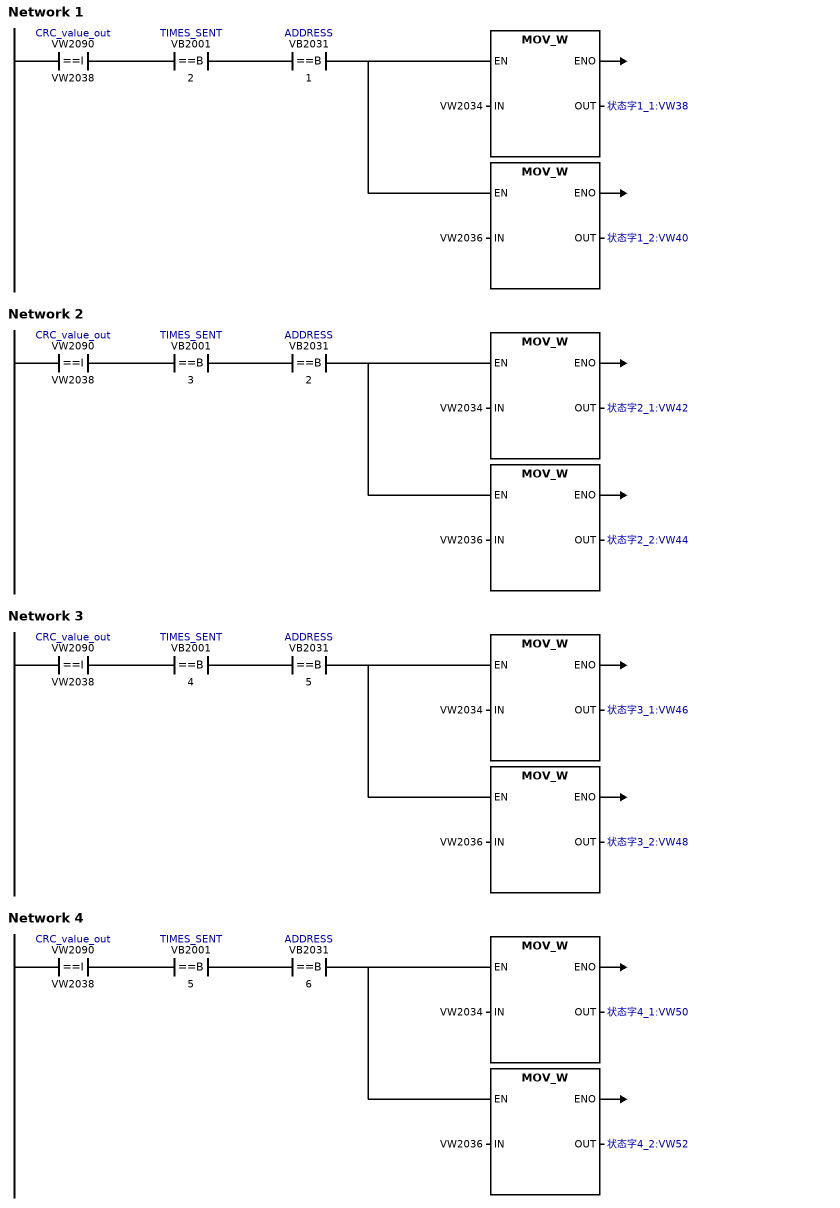
[picture p48: SBR52 networks 1-4]
Network 1
LDW=   CRC_value_out:VW2090, VW2038
AB=    TIMES_SENT:VB2001, 2
AB=    ADDRESS:VB2031, 1
MOVW   VW2034, 状态字1_1:VW38
MOVW   VW2036, 状态字1_2:VW40
Network 2
LDW=   CRC_value_out:VW2090, VW2038
AB=    TIMES_SENT:VB2001, 3
AB=    ADDRESS:VB2031, 2
MOVW   VW2034, 状态字2_1:VW42
MOVW   VW2036, 状态字2_2:VW44
Network 3
LDW=   CRC_value_out:VW2090, VW2038
AB=    TIMES_SENT:VB2001, 4
AB=    ADDRESS:VB2031, 5
MOVW   VW2034, 状态字3_1:VW46
MOVW   VW2036, 状态字3_2:VW48
Network 4
LDW=   CRC_value_out:VW2090, VW2038
AB=    TIMES_SENT:VB2001, 5
AB=    ADDRESS:VB2031, 6
MOVW   VW2034, 状态字4_1:VW50
MOVW   VW2036, 状态字4_2:VW52
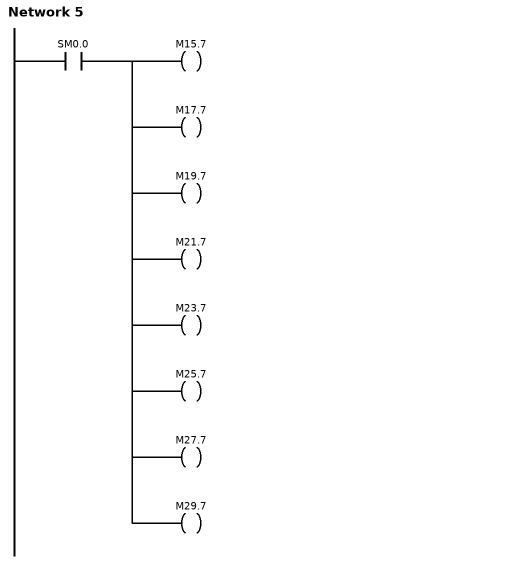
Network 5
LD     SM0.0
=      M15.7
=      M17.7
=      M19.7
=      M21.7
=      M23.7
=      M25.7
=      M27.7
=      M29.7
END_SUBROUTINE_BLOCK

SUBROUTINE_BLOCK COMM_CHECK:SBR53
TITLE=SUBROUTINE COMMENTS
VAR
TEMP1:BOOL;	// L0.0 
TEMP2:BOOL;	// L0.1 
TEMP3:BOOL;	// L0.2 
END_VAR
BEGIN
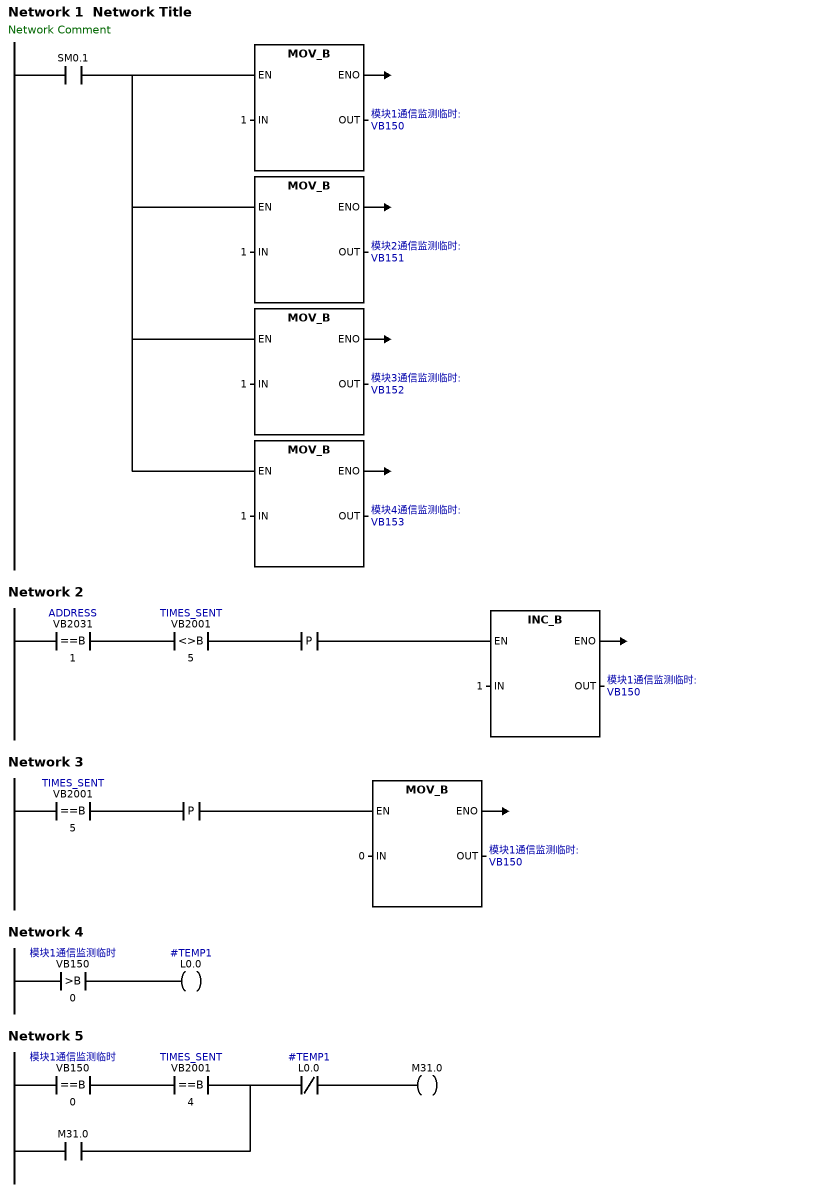
Network 1 // Network Title
// Network Comment
LD     SM0.1
MOVB   1, 模块1通信监测临时:VB150
MOVB   1, 模块2通信监测临时:VB151
MOVB   1, 模块3通信监测临时:VB152
MOVB   1, 模块4通信监测临时:VB153
Network 2
LDB=   ADDRESS:VB2031, 1
AB<>   TIMES_SENT:VB2001, 5
EU
MOVB   1, 模块1通信监测临时:VB150
INCB   模块1通信监测临时:VB150
Network 3
LDB=   TIMES_SENT:VB2001, 5
EU
MOVB   0, 模块1通信监测临时:VB150
Network 4
LDB>   模块1通信监测临时:VB150, 0
=      #TEMP1:L0.0
Network 5
LDB=   模块1通信监测临时:VB150, 0
AB=    TIMES_SENT:VB2001, 4
O      M31.0
AN     #TEMP1:L0.0
=      M31.0
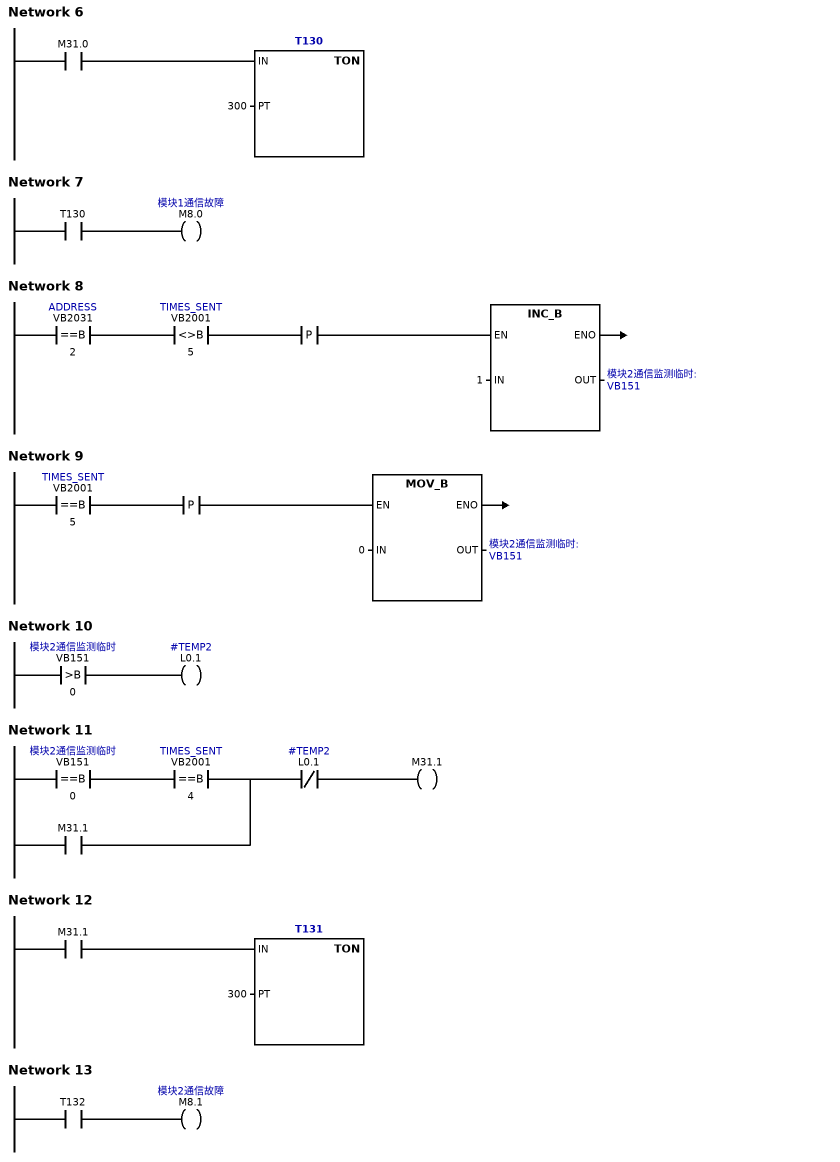
Network 6
LD     M31.0
TON    T130, 300
Network 7
LD     T130
=      模块1通信故障:M8.0
Network 8
LDB=   ADDRESS:VB2031, 2
AB<>   TIMES_SENT:VB2001, 5
EU
MOVB   1, 模块2通信监测临时:VB151
INCB   模块2通信监测临时:VB151
Network 9
LDB=   TIMES_SENT:VB2001, 5
EU
MOVB   0, 模块2通信监测临时:VB151
Network 10
LDB>   模块2通信监测临时:VB151, 0
=      #TEMP2:L0.1
Network 11
LDB=   模块2通信监测临时:VB151, 0
AB=    TIMES_SENT:VB2001, 4
O      M31.1
AN     #TEMP2:L0.1
=      M31.1
Network 12
LD     M31.1
TON    T131, 300
Network 13
LD     T132
=      模块2通信故障:M8.1
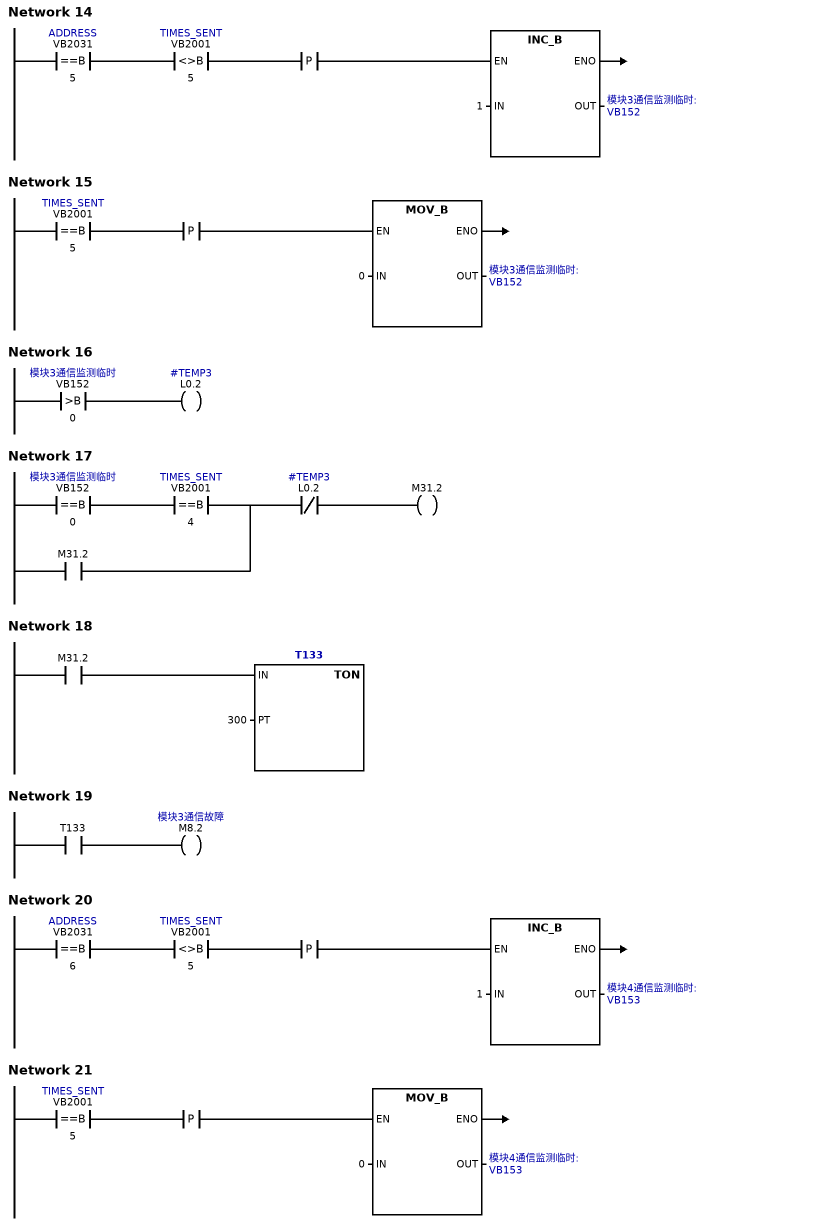
Network 14
LDB=   ADDRESS:VB2031, 5
AB<>   TIMES_SENT:VB2001, 5
EU
MOVB   1, 模块3通信监测临时:VB152
INCB   模块3通信监测临时:VB152
Network 15
LDB=   TIMES_SENT:VB2001, 5
EU
MOVB   0, 模块3通信监测临时:VB152
Network 16
LDB>   模块3通信监测临时:VB152, 0
=      #TEMP3:L0.2
Network 17
LDB=   模块3通信监测临时:VB152, 0
AB=    TIMES_SENT:VB2001, 4
O      M31.2
AN     #TEMP3:L0.2
=      M31.2
Network 18
LD     M31.2
TON    T133, 300
Network 19
LD     T133
=      模块3通信故障:M8.2
Network 20
LDB=   ADDRESS:VB2031, 6
AB<>   TIMES_SENT:VB2001, 5
EU
MOVB   1, 模块4通信监测临时:VB153
INCB   模块4通信监测临时:VB153
Network 21
LDB=   TIMES_SENT:VB2001, 5
EU
MOVB   0, 模块4通信监测临时:VB153
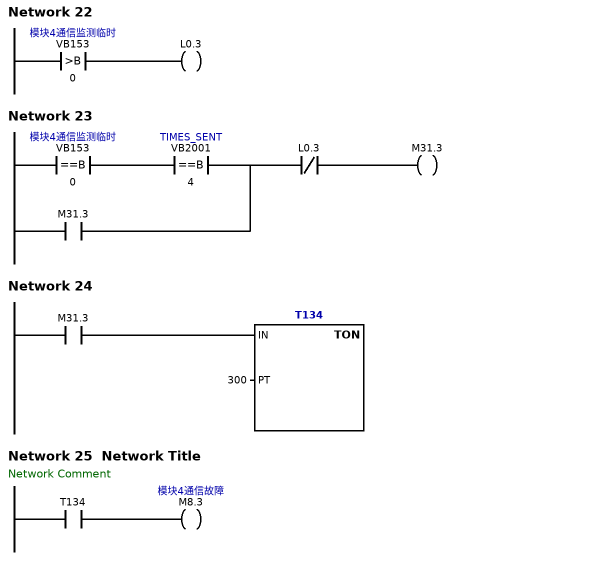
Network 22
LDB>   模块4通信监测临时:VB153, 0
=      L0.3
Network 23
LDB=   模块4通信监测临时:VB153, 0
AB=    TIMES_SENT:VB2001, 4
O      M31.3
AN     L0.3
=      M31.3
Network 24
LD     M31.3
TON    T134, 300
Network 25 // Network Title
// Network Comment
LD     T134
=      模块4通信故障:M8.3
END_SUBROUTINE_BLOCK

SUBROUTINE_BLOCK COMM_ARRAY:SBR54
TITLE=SUBROUTINE COMMENTS
VAR_INPUT
SLAVER_ADR:BYTE;	// LB0 
STAR_REG:BYTE;	// LB1 
REG_LEN:BYTE;	// LB2 
END_VAR
VAR_OUTPUT
ARRAY_T1:WORD;	// LW3 
ARRAY_T2:WORD;	// LW5 
ARRAY_T3:WORD;	// LW7 
ARRAY_T4:WORD;	// LW9 
END_VAR
BEGIN
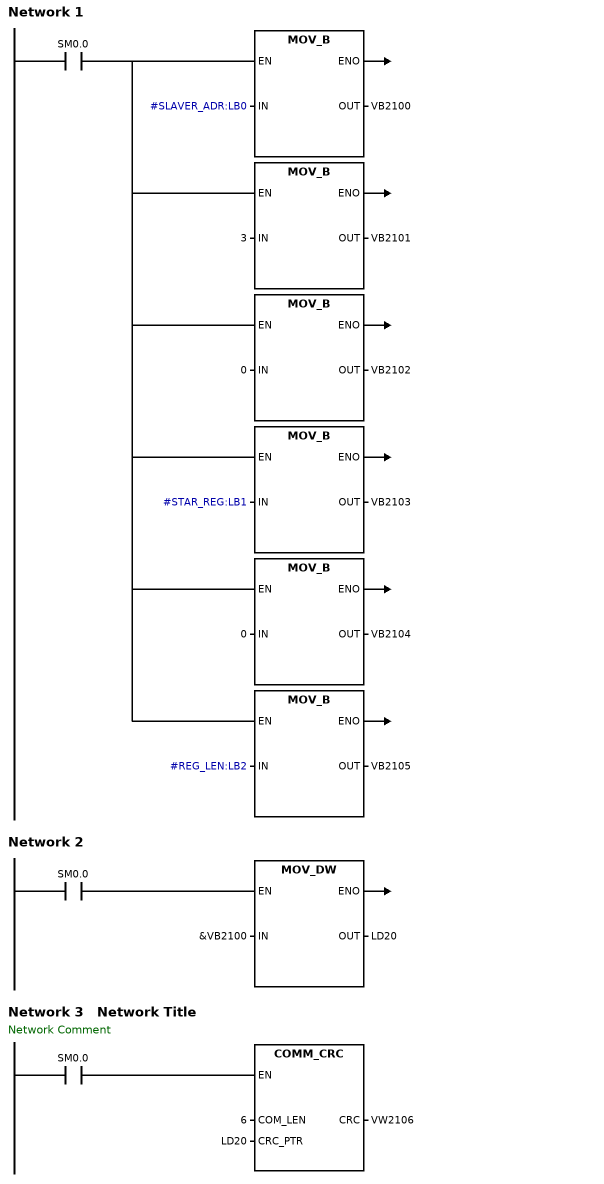
Network 1
LD     SM0.0
MOVB   #SLAVER_ADR:LB0, VB2100
MOVB   3, VB2101
MOVB   0, VB2102
MOVB   #STAR_REG:LB1, VB2103
MOVB   0, VB2104
MOVB   #REG_LEN:LB2, VB2105
Network 2
LD     SM0.0
MOVD   &VB2100, LD20
Network 3 //  Network Title
//  Network Comment
LD     SM0.0
CALL   COMM_CRC:SBR51, 6, LD20, VW2106
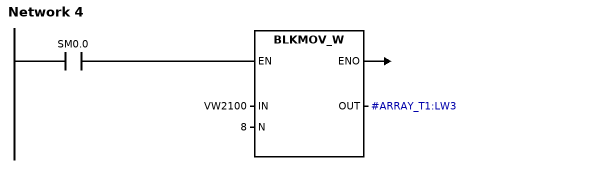
Network 4
LD     SM0.0
BMW    VW2100, #ARRAY_T1:LW3, 8
END_SUBROUTINE_BLOCK

SUBROUTINE_BLOCK PORT_SET:SBR55
TITLE=SUBROUTINE COMMENTS
VAR_INPUT
PORT:BYTE;	// LB0 端口
SPEECH:WORD;	// LW1 通信速率（1200，2400，4800，9600，19200）
DATABIT:BYTE;	// LB3 数据位（7或8）
CHECK:BYTE;	// LB4 是否校验（0：无校验；1：偶校验；2：奇校验）
END_VAR
VAR
ONN:BOOL;	// L5.0 
SETING:BYTE;	// LB6 
TEMP:WORD;	// LW7 
END_VAR
BEGIN
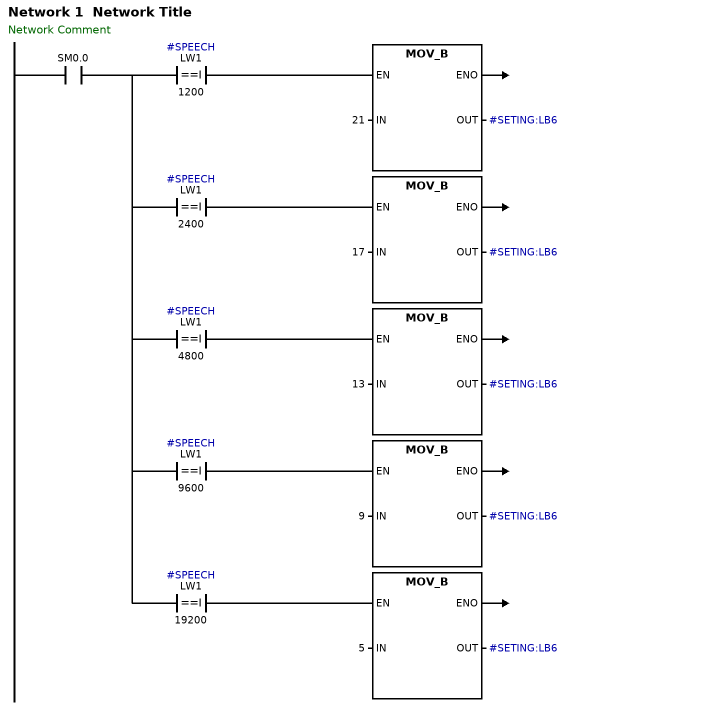
Network 1 // Network Title
// Network Comment
// (network saved uncompiled; LAD cells follow)
// row 0: c0 -| |- SM0.0 v  c1 -|==I|- #SPEECH:LW1, 1200  c2 --  c3 [MOV_B EN:=power@row0, IN:=21, ENO=>power, OUT=>#SETING:LB6]  c4 ->
// row 1: c0 ^v  c3 [box]
// row 2: c0 ^v  c1 -|==I|- #SPEECH:LW1, 2400  c2 --  c3 [MOV_B EN:=power@row2, IN:=17, ENO=>power, OUT=>#SETING:LB6]  c4 ->
// row 3: c0 ^v  c3 [box]
// row 4: c0 ^v  c1 -|==I|- #SPEECH:LW1, 4800  c2 --  c3 [MOV_B EN:=power@row4, IN:=13, ENO=>power, OUT=>#SETING:LB6]  c4 ->
// row 5: c0 ^v  c3 [box]
// row 6: c0 ^v  c1 -|==I|- #SPEECH:LW1, 9600  c2 --  c3 [MOV_B EN:=power@row6, IN:=9, ENO=>power, OUT=>#SETING:LB6]  c4 ->
// row 7: c0 ^v  c3 [box]
// row 8: c0 ^  c1 -|==I|- #SPEECH:LW1, 19200  c2 --  c3 [MOV_B EN:=power@row8, IN:=5, ENO=>power, OUT=>#SETING:LB6]  c4 ->
// row 9: c3 [box]
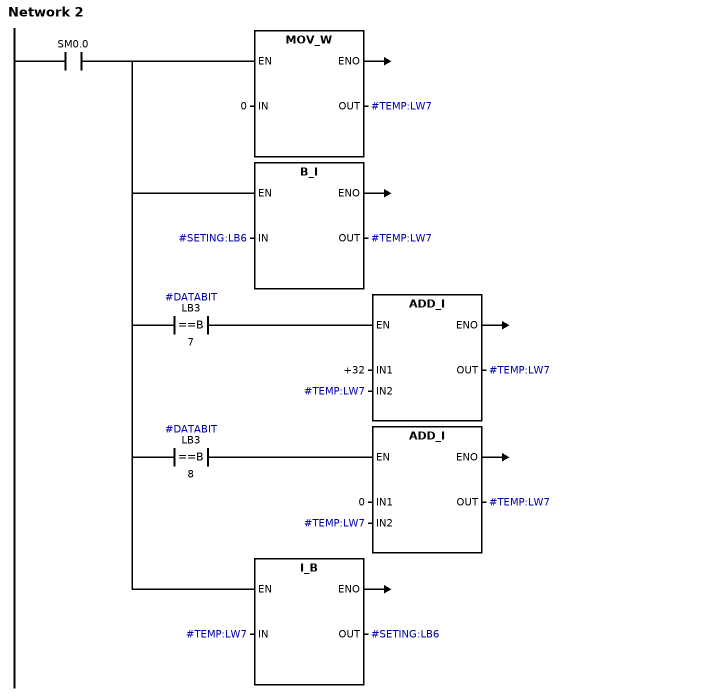
Network 2
// (network saved uncompiled; LAD cells follow)
// row 0: c0 -| |- SM0.0 v  c1 --  c2 [MOV_W EN:=power@row0, IN:=0, ENO=>power, OUT=>#TEMP:LW7]  c3 ->
// row 1: c0 ^v  c2 [box]
// row 2: c0 ^v  c1 --  c2 [B_I EN:=power@row2, IN:=#SETING:LB6, ENO=>power, OUT=>#TEMP:LW7]  c3 ->
// row 3: c0 ^v  c2 [box]
// row 4: c0 ^v  c1 -|==B|- #DATABIT:LB3, 7  c2 --  c3 [ADD_I EN:=power@row4, IN1:=+32, IN2:=#TEMP:LW7, ENO=>power, OUT=>#TEMP:LW7]  c4 ->
// row 5: c0 ^v  c3 [box]
// row 6: c0 ^v  c1 -|==B|- #DATABIT:LB3, 8  c2 --  c3 [ADD_I EN:=power@row6, IN1:=0, IN2:=#TEMP:LW7, ENO=>power, OUT=>#TEMP:LW7]  c4 ->
// row 7: c0 ^v  c3 [box]
// row 8: c0 ^  c1 --  c2 [I_B EN:=power@row8, IN:=#TEMP:LW7, ENO=>power, OUT=>#SETING:LB6]  c3 ->
// row 9: c2 [box]
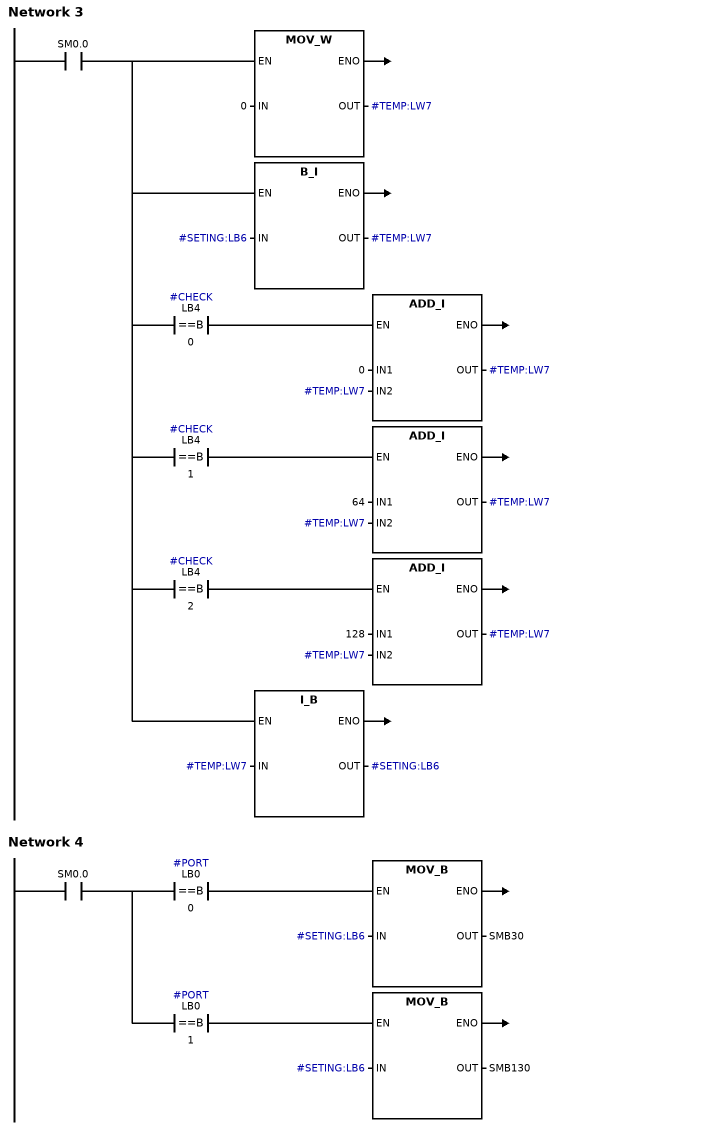
Network 3
// (network saved uncompiled; LAD cells follow)
// row 0: c0 -| |- SM0.0 v  c1 --  c2 [MOV_W EN:=power@row0, IN:=0, ENO=>power, OUT=>#TEMP:LW7]  c3 ->
// row 1: c0 ^v  c2 [box]
// row 2: c0 ^v  c1 --  c2 [B_I EN:=power@row2, IN:=#SETING:LB6, ENO=>power, OUT=>#TEMP:LW7]  c3 ->
// row 3: c0 ^v  c2 [box]
// row 4: c0 ^v  c1 -|==B|- #CHECK:LB4, 0  c2 --  c3 [ADD_I EN:=power@row4, IN1:=0, IN2:=#TEMP:LW7, ENO=>power, OUT=>#TEMP:LW7]  c4 ->
// row 5: c0 ^v  c3 [box]
// row 6: c0 ^v  c1 -|==B|- #CHECK:LB4, 1  c2 --  c3 [ADD_I EN:=power@row6, IN1:=64, IN2:=#TEMP:LW7, ENO=>power, OUT=>#TEMP:LW7]  c4 ->
// row 7: c0 ^v  c3 [box]
// row 8: c0 ^v  c1 -|==B|- #CHECK:LB4, 2  c2 --  c3 [ADD_I EN:=power@row8, IN1:=128, IN2:=#TEMP:LW7, ENO=>power, OUT=>#TEMP:LW7]  c4 ->
// row 9: c0 ^v  c3 [box]
// row 10: c0 ^  c1 --  c2 [I_B EN:=power@row10, IN:=#TEMP:LW7, ENO=>power, OUT=>#SETING:LB6]  c3 ->
// row 11: c2 [box]
Network 4
// (network saved uncompiled; LAD cells follow)
// row 0: c0 -| |- SM0.0 v  c1 -|==B|- #PORT:LB0, 0  c2 --  c3 [MOV_B EN:=power@row0, IN:=#SETING:LB6, ENO=>power, OUT=>SMB30]  c4 ->
// row 1: c0 ^v  c3 [box]
// row 2: c0 ^  c1 -|==B|- #PORT:LB0, 1  c2 --  c3 [MOV_B EN:=power@row2, IN:=#SETING:LB6, ENO=>power, OUT=>SMB130]  c4 ->
// row 3: c3 [box]
END_SUBROUTINE_BLOCK

SUBROUTINE_BLOCK MES_SEND:SBR56
TITLE=SUBROUTINE COMMENTS
BEGIN
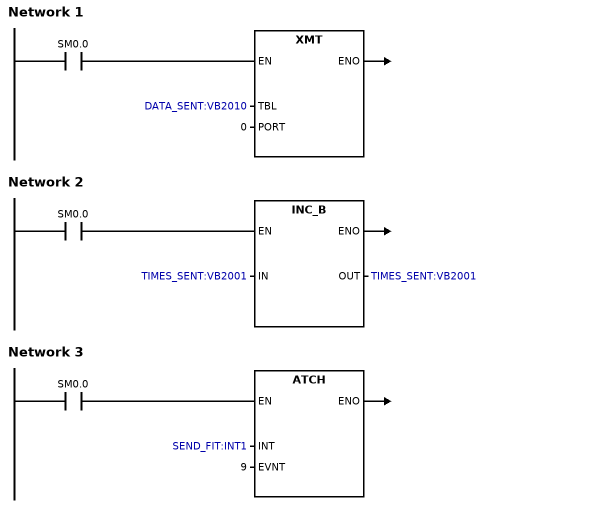
Network 1 // 
	
LD     SM0.0
XMT    DATA_SENT:VB2010, 0
Network 2
LD     SM0.0
INCB   TIMES_SENT:VB2001
Network 3
LD     SM0.0
ATCH   SEND_FIT:INT1, 9
Network 4 // Network Title
// Network Comment
END_SUBROUTINE_BLOCK

SUBROUTINE_BLOCK ARRAY_INSTR:SBR60
TITLE=旧的4块镇流器监测模块的地址分别是1,2,3,5
BEGIN
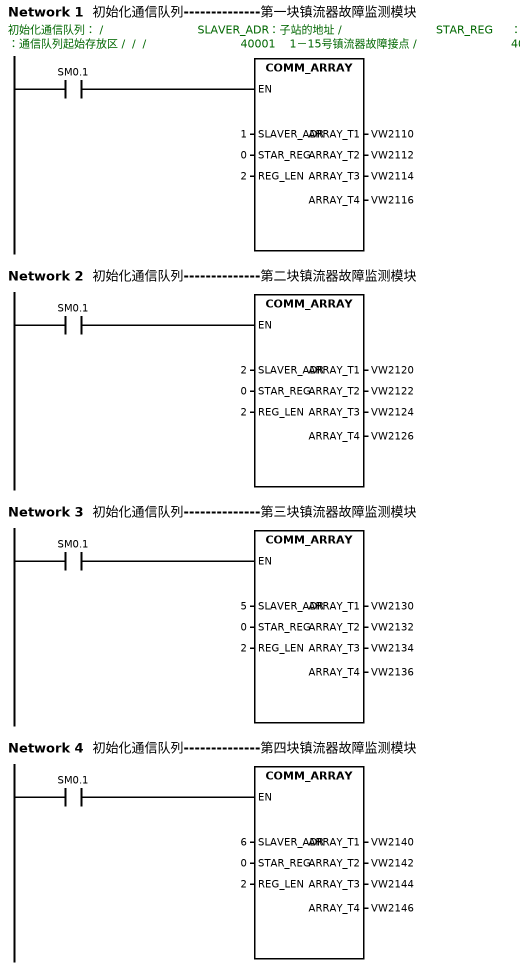
Network 1 // 初始化通信队列--------------第一块镇流器故障监测模块
// 初始化通信队列：
//                           SLAVER_ADR：子站的地址
//                           STAR_REG     ：子站数据起始寄存器
//                           REG_LEN        ：读取的数据寄存器长度
//                           ARRAY_T        ：通信队列起始存放区
// 
// 
//                           40001		1－15号镇流器故障接点
//                           40002		16－30号镇流器故障接点
//                         
LD     SM0.1
CALL   COMM_ARRAY:SBR54, 1, 0, 2, VW2110, VW2112, VW2114, VW2116
Network 2 // 初始化通信队列--------------第二块镇流器故障监测模块
LD     SM0.1
CALL   COMM_ARRAY:SBR54, 2, 0, 2, VW2120, VW2122, VW2124, VW2126
Network 3 // 初始化通信队列--------------第三块镇流器故障监测模块
LD     SM0.1
CALL   COMM_ARRAY:SBR54, 5, 0, 2, VW2130, VW2132, VW2134, VW2136
Network 4 // 初始化通信队列--------------第四块镇流器故障监测模块
LD     SM0.1
CALL   COMM_ARRAY:SBR54, 6, 0, 2, VW2140, VW2142, VW2144, VW2146
END_SUBROUTINE_BLOCK

INTERRUPT_BLOCK DATA_READ:INT0
TITLE=
BEGIN
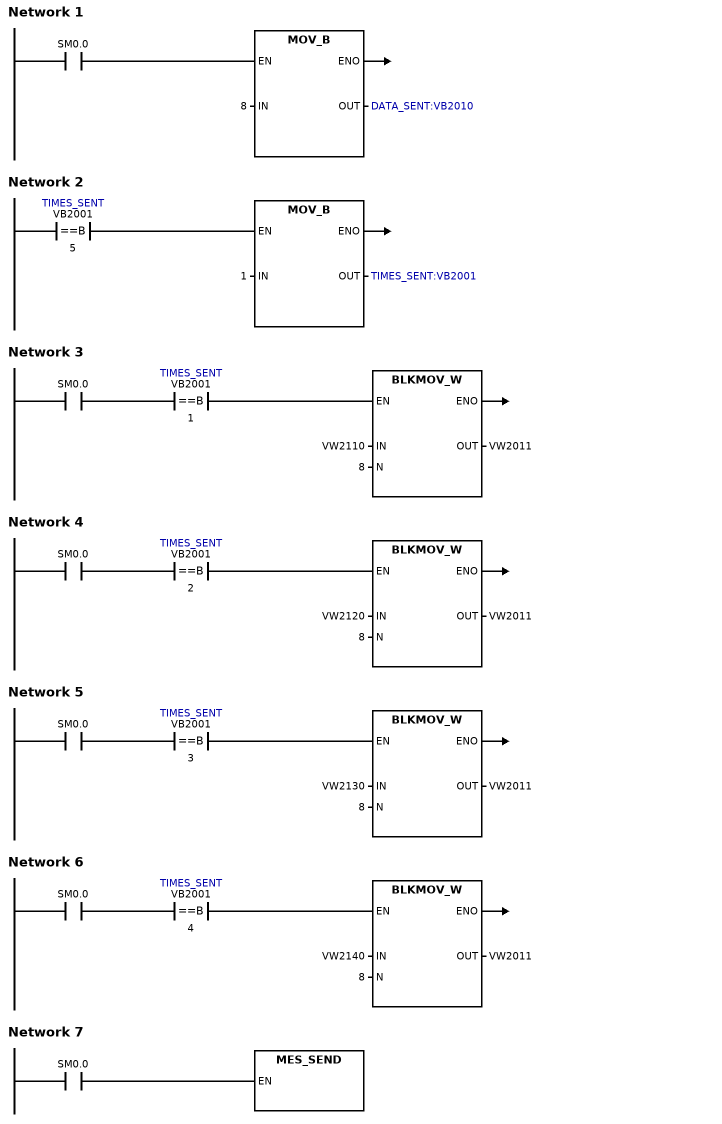
Network 1
// (network saved uncompiled; LAD cells follow)
// row 0: c0 -| |- SM0.0  c1 --  c2 [MOV_B EN:=power@row0, IN:=8, ENO=>power, OUT=>DATA_SENT:VB2010]  c3 ->
// row 1: c2 [box]
Network 2
// (network saved uncompiled; LAD cells follow)
// row 0: c0 -|==B|- TIMES_SENT:VB2001, 5  c1 --  c2 [MOV_B EN:=power@row0, IN:=1, ENO=>power, OUT=>TIMES_SENT:VB2001]  c3 ->
// row 1: c2 [box]
Network 3
// (network saved uncompiled; LAD cells follow)
// row 0: c0 -| |- SM0.0  c1 -|==B|- TIMES_SENT:VB2001, 1  c2 --  c3 [BLKMOV_W EN:=power@row0, IN:=VW2110, N:=8, ENO=>power, OUT=>VW2011]  c4 ->
// row 1: c3 [box]
Network 4
// (network saved uncompiled; LAD cells follow)
// row 0: c0 -| |- SM0.0  c1 -|==B|- TIMES_SENT:VB2001, 2  c2 --  c3 [BLKMOV_W EN:=power@row0, IN:=VW2120, N:=8, ENO=>power, OUT=>VW2011]  c4 ->
// row 1: c3 [box]
Network 5
// (network saved uncompiled; LAD cells follow)
// row 0: c0 -| |- SM0.0  c1 -|==B|- TIMES_SENT:VB2001, 3  c2 --  c3 [BLKMOV_W EN:=power@row0, IN:=VW2130, N:=8, ENO=>power, OUT=>VW2011]  c4 ->
// row 1: c3 [box]
Network 6
// (network saved uncompiled; LAD cells follow)
// row 0: c0 -| |- SM0.0  c1 -|==B|- TIMES_SENT:VB2001, 4  c2 --  c3 [BLKMOV_W EN:=power@row0, IN:=VW2140, N:=8, ENO=>power, OUT=>VW2011]  c4 ->
// row 1: c3 [box]
Network 7
// (network saved uncompiled; LAD cells follow)
// row 0: c0 -| |- SM0.0  c1 --  c2 [MES_SEND EN:=power@row0]
END_INTERRUPT_BLOCK

INTERRUPT_BLOCK SEND_FIT:INT1
TITLE=
BEGIN
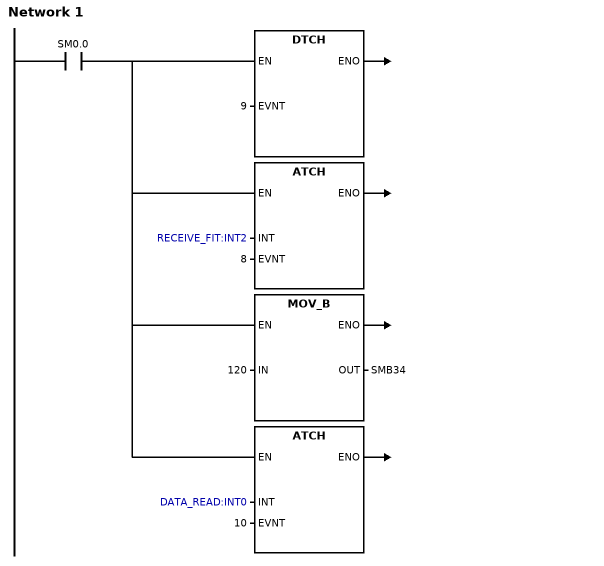
Network 1
LD     SM0.0
DTCH   9
ATCH   RECEIVE_FIT:INT2, 8
MOVB   120, SMB34
ATCH   DATA_READ:INT0, 10
END_INTERRUPT_BLOCK

INTERRUPT_BLOCK RECEIVE_FIT:INT2
TITLE=
BEGIN
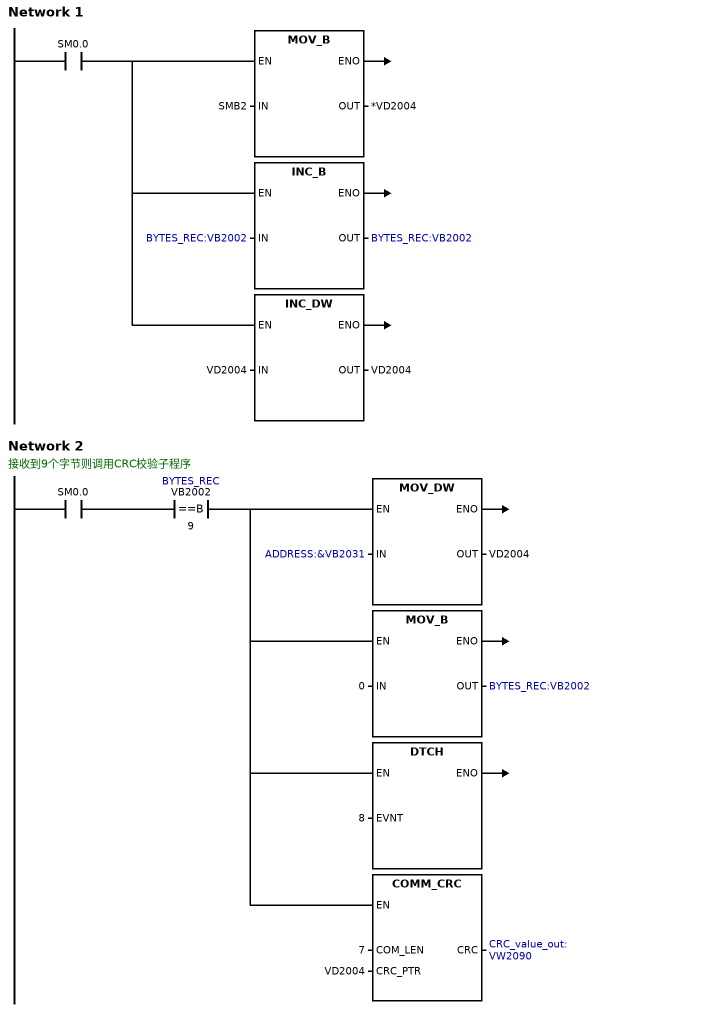
Network 1
// (network saved uncompiled; LAD cells follow)
// row 0: c0 -| |- SM0.0 v  c1 --  c2 [MOV_B EN:=power@row0, IN:=SMB2, ENO=>power, OUT=>*VD2004]  c3 ->
// row 1: c0 ^v  c2 [box]
// row 2: c0 ^v  c1 --  c2 [INC_B EN:=power@row2, IN:=BYTES_REC:VB2002, ENO=>power, OUT=>BYTES_REC:VB2002]  c3 ->
// row 3: c0 ^v  c2 [box]
// row 4: c0 ^  c1 --  c2 [INC_DW EN:=power@row4, IN:=VD2004, ENO=>power, OUT=>VD2004]  c3 ->
// row 5: c2 [box]
Network 2
// 接收到9个字节则调用CRC校验子程序 
// (network saved uncompiled; LAD cells follow)
// row 0: c0 -| |- SM0.0  c1 -|==B|- BYTES_REC:VB2002, 9 v  c2 --  c3 [MOV_DW EN:=power@row0, IN:=&ADDRESS:VB2031, ENO=>power, OUT=>VD2004]  c4 ->
// row 1: c1 ^v  c3 [box]
// row 2: c1 ^v  c2 --  c3 [MOV_B EN:=power@row2, IN:=0, ENO=>power, OUT=>BYTES_REC:VB2002]  c4 ->
// row 3: c1 ^v  c3 [box]
// row 4: c1 ^v  c2 --  c3 [DTCH EN:=power@row4, EVNT:=8, ENO=>power]  c4 ->
// row 5: c1 ^v  c3 [box]
// row 6: c1 ^  c2 --  c3 [COMM_CRC EN:=power@row6, COM_LEN:=7, CRC_PTR:=VD2004, CRC=>CRC_value_out:VW2090]
// row 7: c3 [box]
END_INTERRUPT_BLOCK
